FUNCTION_BLOCK TmsEmbarkStation EXTENDS Process IMPLEMENTS ITF_SwitchStation
VAR
	DepartMover : ITmsMover;
	_StateMachine : IPmlStateMachine;
	_TmsSwitch : ITF_TmsSwitch;
	_TrackLevel : INT := 1; //1 is low, 2 is high
	State :(
		Init,                                               
		Ready,                                 
        Waiting,
		HasSwitch,
		Call,
		Processing,
		Boarding,
		BoardingComplete,
		Moving,
		Aborting); 
	_switchPosition: MC_LREAL;
	demandPosition : TmsSwitchPosition;
	arrTrackIds : ARRAY[1..4] OF OTCID;
	isUpAllowed : BOOL := TRUE;
	isDownAllowed : BOOL := FALSE;
	isMiddleAllowed : BOOL := TRUE;
	_BoardVelocity : MC_LREAL;
END_VAR

{analysis -2}

PROPERTY BoardVelocity : MC_LREAL
GET
BoardVelocity := _BoardVelocity;
END_GET
SET
_BoardVelocity := BoardVelocity;
END_SET
END_PROPERTY

METHOD PUBLIC  Cycle : HRESULT
VAR_INPUT
END_VAR
CASE State OF
	Init:
		_Operating := _Clear := _Complete := _Ready := _HasMover := FALSE;
		StationMovers := 0;
		State := Ready;
	
	Ready:	
		IF _StateMachine.GetCurrentState() = E_PMLState.ePMLState_Clearing THEN
			_Operating := _Complete := _HasMover := FALSE;
			_Clear := _Ready := TRUE;
			StationMovers := 0;
			State := Waiting;
		END_IF
		IF _StateMachine.GetCurrentState() = E_PMLState.ePMLState_Aborting THEN
			State := Aborting;
		END_IF
	
	Waiting:
		IF _HasMover THEN
			State := HasSwitch;
			_Operating := TRUE;
			_Clear := FALSE;
			_Ready := FALSE;
			_Complete := FALSE;
		END_IF
		IF _StateMachine.GetCurrentState() = E_PMLState.ePMLState_Aborting THEN
			State := Aborting;
		END_IF
	
	HasSwitch:
		IF (_TrackLevel = 1 AND (TmsSwitch.Switch = TmsSwitchPosition.Down OR (TmsSwitch.Switch = TmsSwitchPosition.Middle AND isUpAllowed)))
			OR (_TrackLevel = 2 AND (TmsSwitch.Switch = TmsSwitchPosition.Up OR (TmsSwitch.Switch = TmsSwitchPosition.Middle AND isDownAllowed))) THEN
				IF TmsSwitch.ExchangeMover(Mover := DepartMover, currentStation := THIS^) THEN
					State := Processing;
				END_IF
		ELSE
			State := Call;
		END_IF
		IF _StateMachine.GetCurrentState() = E_PMLState.ePMLState_Aborting THEN
			State := Aborting;
		END_IF	
		
	Call:
		IF NOT TmsSwitch.HasMover() AND TmsSwitch.IsStationary() THEN
			IF TmsSwitch.MoveTo(positionState := TmsSwitchPosition.Middle) THEN
				State := HasSwitch;
			END_IF
		ELSE
			State := Waiting;
		END_IF
		IF _StateMachine.GetCurrentState() = E_PMLState.ePMLState_Aborting THEN
			State := Aborting;
		END_IF
	
	Processing:
		IF _TrackLevel = 1 THEN
			IF TmsSwitch.Switch = TmsSwitchPosition.Down and isMiddleAllowed THEN
				IF DepartMover.ActiveTrack = arrTrackIds[4] THEN
					State := Boarding;
				ELSE
					DepartMover.ActivateTrack(arrTrackIds[4]);
					State := Boarding;
				END_IF
				demandPosition := TmsSwitchPosition.Middle;
			ELSIF TmsSwitch.Switch = TmsSwitchPosition.Middle AND isUpAllowed THEN
				IF DepartMover.ActiveTrack = arrTrackIds[1] THEN
					State := Boarding;
				ELSE
					DepartMover.ActivateTrack(arrTrackIds[1]);
					State := Boarding;
				END_IF
				demandPosition := TmsSwitchPosition.Up;
			END_IF
		ELSE
			IF TmsSwitch.Switch = TmsSwitchPosition.Up AND isMiddleAllowed THEN
				IF DepartMover.ActiveTrack = arrTrackIds[3] THEN
					State := Boarding;
				ELSE
					DepartMover.ActivateTrack(arrTrackIds[3]);
					State := Boarding;
				END_IF
				demandPosition := TmsSwitchPosition.Middle;
			ELSIF TmsSwitch.Switch = TmsSwitchPosition.Middle AND isDownAllowed THEN
				IF DepartMover.ActiveTrack = arrTrackIds[2] THEN
					State := Boarding;
				ELSE
					DepartMover.ActivateTrack(arrTrackIds[2]);
					State := Boarding;
				END_IF
				demandPosition := TmsSwitchPosition.Down;
			END_IF
		END_IF
		IF _StateMachine.GetCurrentState() = E_PMLState.ePMLState_Aborting THEN
			State := Aborting;
		END_IF
		
	Boarding:
		DepartMover.MoveTo(Position := _switchPosition, Velocity := _BoardVelocity, BackwardMove := FALSE);
		IF DepartMover.isAtPosition(position := _switchPosition) THEN
			State := BoardingComplete;
		END_IF
		
	BoardingComplete:
		IF TmsSwitch.MoveTo(positionState := demandPosition) THEN
			State := Moving;
		END_IF
		IF _StateMachine.GetCurrentState() = E_PMLState.ePMLState_Aborting THEN
			State := Aborting;
		END_IF
		
	Moving:
		IF _Complete AND NOT _HasMover THEN
			_Operating := FALSE;
			_Clear := TRUE;
			_Ready := TRUE;
			State := Waiting;
		END_IF
		IF _StateMachine.GetCurrentState() = E_PMLState.ePMLState_Aborting THEN
			State := Aborting;
		END_IF	

	Aborting:
		State := Ready;	
		DepartMover := 0;
END_CASE
SUPER^.Cycle();
Cycle := S_OK;
END_METHOD

METHOD HasMover : BOOL
VAR_INPUT
	mover : IMover;
END_VAR
VAR
	iTmsMover : ITmsMover;
END_VAR
IF StationMovers <= 2 THEN
	StationMovers := StationMovers + 1;
	IF __QUERYINTERFACE(mover,iTmsMover) THEN
		DepartMover := iTmsMover;
		_HasMover := true;
	END_IF
END_IF
HasMover := TRUE;
END_METHOD

METHOD PUBLIC MoverAway : BOOL
VAR_INPUT
END_VAR
StationMovers := StationMovers - 1;
IF StationMovers = 0 THEN
	_HasMover := FALSE;
END_IF
DepartMover := 0;
END_METHOD

PROPERTY PmlStateMachine : IPmlStateMachine
GET
PmlStateMachine := _StateMachine;
END_GET
SET
_StateMachine := PmlStateMachine;
END_SET
END_PROPERTY

METHOD PUBLIC SwitchMoveComplete : BOOL
VAR_INPUT
END_VAR
_Complete := SwitchMoveComplete := true;
END_METHOD

PROPERTY SwitchTravelPosition : mc_lreal
GET
SwitchTravelPosition := _switchPosition;
END_GET
SET
_switchPosition := SwitchTravelPosition;
END_SET
END_PROPERTY

PROPERTY TmsSwitch : ITF_TmsSwitch
GET
TmsSwitch := _TmsSwitch;
END_GET
SET
_TmsSwitch := TmsSwitch;
END_SET
END_PROPERTY

PROPERTY TrackIds : array[1..4] of otcid
GET
TrackIds := arrTrackIds;
END_GET
SET
arrTrackIds := TrackIds;
END_SET
END_PROPERTY

PROPERTY TrackLevel : INT
GET
TrackLevel := _TrackLevel;
END_GET
SET
_TrackLevel := TrackLevel;
END_SET
END_PROPERTY

END_FUNCTION_BLOCK

(* stored: Version 1.1.0.1, ProductVersion 3.1.4024.12
   POU TmsEmbarkStation: Id {4d15a973-29cb-4ffe-934a-8f072d992ec0}, SpecialFunc None
   Property BoardVelocity: Id {af5577ef-90f6-4070-9e3d-dce62d068c94}
   Get Get: Id {442f20d9-4d5c-462e-ace0-37721614361e}
   Set Set: Id {4f476cb8-1c36-46ee-b33f-8098bec190be}
   Method Cycle: Id {30dc7518-cfa1-45c8-85d7-d03d0ef4ae28}
   Method HasMover: Id {466b4750-cbf0-42df-80f2-b3d4852756ba}
   Method MoverAway: Id {45498adf-6827-4a97-8c80-ff53aebb1724}
   Property PmlStateMachine: Id {a47db168-d2a9-4247-adb9-892ae103948e}
   Get Get: Id {7455cd11-5ef8-425b-8f7e-20b1eaa44250}
   Set Set: Id {70867ab3-cb45-4255-9352-18cd1c4ce7ec}
   Method SwitchMoveComplete: Id {a8eedfd9-7707-47a4-b55d-1e335fa7f41f}
   Property SwitchTravelPosition: Id {506615ae-e584-4b6b-8c90-23702c945ca0}
   Get Get: Id {770e482e-e926-4e26-8349-fb06dc2d74be}
   Set Set: Id {2f71d79c-8b57-4fda-9b2a-e631ae1faffd}
   Property TmsSwitch: Id {32709822-da92-40fc-979a-5a9084ca9dfd}
   Get Get: Id {afd06df8-55b5-473c-ad0b-a2b8f0614d91}
   Set Set: Id {afdc9e35-5be9-439b-973f-2fdfa7b2941c}
   Property TrackIds: Id {5077a096-7fe1-4a0a-87f3-6619fda26f3f}
   Get Get: Id {b5bca1f7-f5d0-4d03-9e76-4e8c0b77044c}
   Set Set: Id {bdbe3d16-cad0-4d02-9f21-8379c823a76d}
   Property TrackLevel: Id {3cbcc021-27ff-4251-b3d2-761cf34c192e}
   Get Get: Id {eac07d3d-cc95-4d94-be8d-aab0ced9fdea}
   Set Set: Id {4b1478e4-977e-454a-a0bf-fe888f795dfb} *)
